(* PLC project v0.6.02_RefactorGateAndTest.project, CODESYS CODESYS V3.5 SP19 Patch 1 *)
(* stored: creationDateTime 2026-08-11T18:19:14.785911, modificationDateTime 2026-08-11T18:19:14.785911 *)

(* ============================================================== [IHM] ST_Safety_Emergency_HmiCmd -- Commandes IHM pour la chaine AU -------------------------------------------------------------- Role : structure d'echange pour les commandes operateur de la chaine d'arret d'urgence (miroir ST_ModesCmd). Pattern : identique a GVL_IHM.Modes.Cmd dans le projet reel. L'IHM ecrit ces champs, le programme les consomme. ============================================================== Docs : DOC/AF/AF_Partie-01_Analyse_Fonctionnelle_v2.0.md DOC/AF/AF_Partie-07_Interface_IHM_v2.0.md *)
TYPE ST_Safety_Emergency_HmiCmd : STRUCT
  BtnEmergencyArming : BOOL;  (* Front demande rearmement contacteur *)
  BtnEmergencyCutOff : BOOL;  (* Niveau coupure IHM maintenue *)
  BtnFaultReset : BOOL;  (* Front acquittement defauts *)
END_STRUCT;
END_TYPE
